FUNCTION_BLOCK FB_System_LA_955
VAR_INPUT
	Betrieb_Anford_auto		: BOOL;
	Freigabe_auto			: BOOL;
	FBT_Zustand				: ST_System_FBT_Zustand; (* Zustand Fußbodentemperierung *)
END_VAR
VAR_OUTPUT
END_VAR
VAR
	{attribute 'OPC.UA.DA' := '1'}Zustand					: ST_System_LA_Zustand;	
	{attribute 'OPC.UA.DA' := '1'}Parameter				: ST_System_LA_Parameter;	
	Stellwert				: ST_System_LA_Stellwert;

	Stellventil_453			: FB_SVs;
	Stellventil_454			: FB_SVs;
	Pumpe_455				: FB_PU_les;
	Regelventil_455			: FB_RV_les;
	Lueftungsanlage_955		: FB_LA;

	Zustandscheck			: FB_System_LA_Zustandscheck;
END_VAR

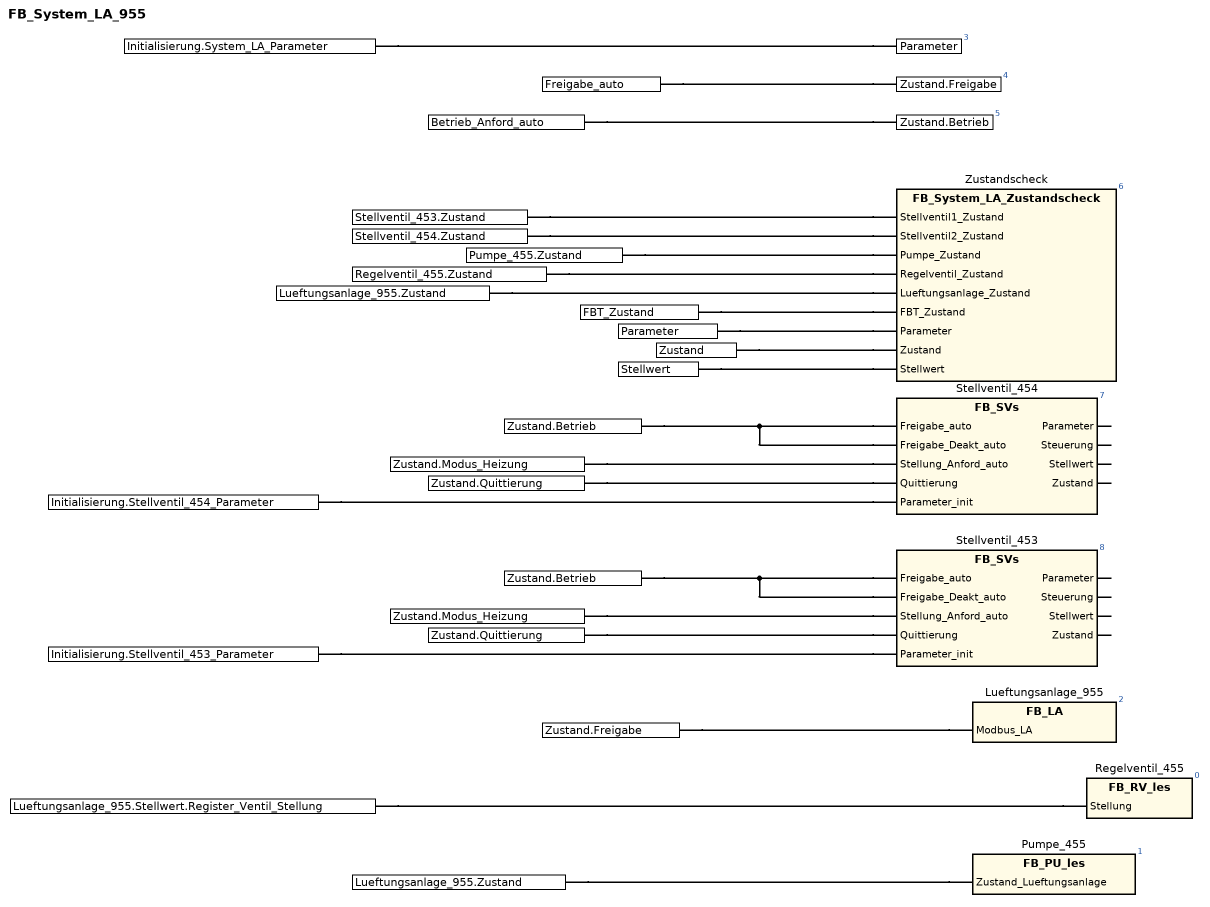
Regelventil_455(Stellung := Lueftungsanlage_955.Stellwert.Register_Ventil_Stellung); // FB_RV_les
Pumpe_455(Zustand_Lueftungsanlage := Lueftungsanlage_955.Zustand); // FB_PU_les
Lueftungsanlage_955(Modbus_LA := Zustand.Freigabe); // FB_LA
Parameter := Initialisierung.System_LA_Parameter;
Zustand.Freigabe := Freigabe_auto;
Zustand.Betrieb := Betrieb_Anford_auto;
Zustandscheck(
    Stellventil1_Zustand := Stellventil_453.Zustand,
    Stellventil2_Zustand := Stellventil_454.Zustand,
    Pumpe_Zustand := Pumpe_455.Zustand,
    Regelventil_Zustand := Regelventil_455.Zustand,
    Lueftungsanlage_Zustand := Lueftungsanlage_955.Zustand,
    FBT_Zustand := FBT_Zustand,
    Parameter := Parameter,
    Zustand := Zustand,
    Stellwert := Stellwert); // FB_System_LA_Zustandscheck
Stellventil_454(
    Freigabe_auto := Zustand.Betrieb,
    Freigabe_Deakt_auto := Zustand.Betrieb,
    Stellung_Anford_auto := Zustand.Modus_Heizung,
    Quittierung := Zustand.Quittierung,
    Parameter_init := Initialisierung.Stellventil_454_Parameter); // FB_SVs
Stellventil_453(
    Freigabe_auto := Zustand.Betrieb,
    Freigabe_Deakt_auto := Zustand.Betrieb,
    Stellung_Anford_auto := Zustand.Modus_Heizung,
    Quittierung := Zustand.Quittierung,
    Parameter_init := Initialisierung.Stellventil_453_Parameter); // FB_SVs

END_FUNCTION_BLOCK

(* stored: Version 1.1.0.1, ProductVersion 3.1.4024.9
   POU FB_System_LA_955: Id {63cffb3f-4492-4015-9c2e-76831bc53ea7}, SpecialFunc None *)
